DATA_BLOCK "!!instanceOf-CabState$$"
{ S7_Optimized_Access := 'TRUE' }
VERSION : 0.1
NON_RETAIN
"CabState"

BEGIN

END_DATA_BLOCK

